(* PLC project Tc2_System.LPTSIGNAL Demo, tc3-libraries-kb TwinCAT 3.1 *)
(* stored: creationDateTime 2026-05-20T00:00:00, modificationDateTime 2026-05-20T00:00:00 *)

PROGRAM P_Demo_LPTSIGNAL
  VAR
    bLptOk1 : BOOL;  (* 入口拉高调用结果 *)
    bLptOk2 : BOOL;  (* 出口拉低调用结果 *)
  END_VAR

// =============================================================================
// 场景：用示波器观察 MAIN 任务实际周期：入口拉高 D7、出口拉低 D7，示波器看到的方波周期 = 实际任务周期。
// 价值：硬件级时序观察，比日志统计精度高。
// 验证：示波器接 LPT1 D7 引脚 → 看到周期性方波；周期与 SYSTEM 配的任务周期一致。
// 验证步骤：
//   1. 右键 PLC 项目 → Import PLCopenXML → 选本文件
//   2. 引用 Tc2_System（References → Add library）
//   3. 编译 → 登录 → 运行；按上方『验证』行的指示在线写值观察
// =============================================================================

// MAIN 入口拉高 LPT D7 引脚
bLptOk1 := LPTSIGNAL(
    PortAddr := 16#378,
    PinNo    := 7,
    OnOff    := TRUE
);

// ... 此处写业务逻辑（被示波器观察） ...

// MAIN 出口拉低
bLptOk2 := LPTSIGNAL(
    PortAddr := 16#378,
    PinNo    := 7,
    OnOff    := FALSE
);
END_PROGRAM
